// Mitsubishi GX Works2 project: Class2_SelfHolding&InterLock   PLC: Q03UD

PROGRAM MAIN
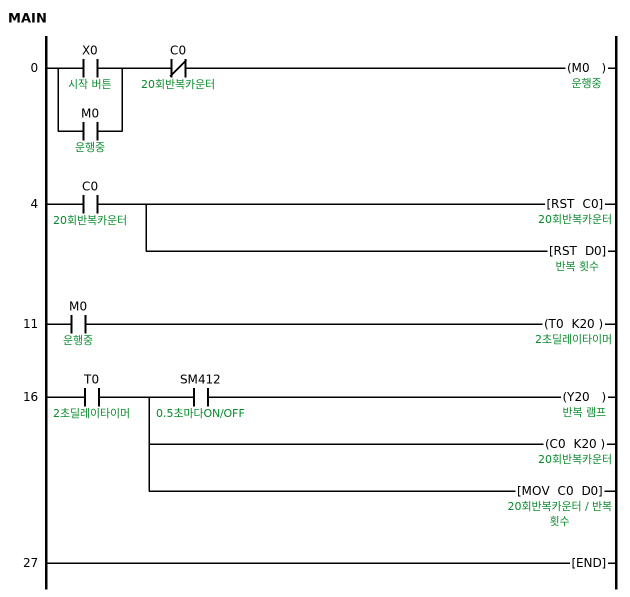
0     LD      X0  ; 시작 버튼
      OR      M0  ; 운행중
      ANI     C0  ; 20회반복카운터
      OUT     M0  ; 운행중
4     LD      C0  ; 20회반복카운터
      RST     C0  ; 20회반복카운터
      RST     D0  ; 반복 횟수
11    LD      M0  ; 운행중
      OUT     T0 K20  ; 2초딜레이타이머
16    LD      T0  ; 2초딜레이타이머
      MPS
      AND     SM412  ; 0.5초마다ON/OFF
      OUT     Y20  ; 반복 램프
      MPP
      OUT     C0 K20  ; 20회반복카운터
      MOV     C0 D0
27    END
END_PROGRAM
